                // --- STATE_NEXT folded into this scan (2026-09-02) --------------
                // Saves one PLC scan per recipe line: the line advance no longer
                // costs its own scan. Body is identical to state 60, which STAYS in
                // place -- ten other states still transition to it.
                //
                // MUST stay below the Error / tonMoveTimeout block above, and MUST
                // keep the #state = STATE_NEXT guard: those branches write
                // STATE_ERROR, and the guard is what lets them win. Removing either
                // makes a faulted axis advance the line instead of stopping.
                // See docs/RecipeHandler_ScanLatency.md.
                IF #state = STATE_NEXT THEN
                    #lineIndex := #lineIndex + 1;
                    IF "DB_HMI".SingleStepMode THEN
                        #state := STATE_STEP_WAIT;
                    ELSE
                        #state := STATE_READ;
                    END_IF;
                END_IF;
            END_IF;

        // -----------------------------------------------------------------
        // === STATE_VEL_WAIT (32) -- EXPERIMENTAL velocity-mode segment ===
        // -----------------------------------------------------------------
        // The axes are moving under MC_MoveVelocity toward #targX/#targZ. Nothing
        // here ends in v = 0: when the remaining distance drops under vmSwitchDist
        // the line is counted done and STATE_READ launches the next one (EXEC
        // computes its vector from the ACTUAL position, so the lag of that scan is
        // corrected on the next segment instead of accumulating).
        //
        // Guard order matters: Pause first (operator intent), then run permission,
        // then faults, then completion. Every exit except completion drops
        // vmActive AND brings in a halt, because MC_MoveVelocity keeps running
        // when Execute drops.
        //
        // Fault exits set vmHaltReq THEMSELVES (2026-09-15). "Going to STATE_ERROR"
        // is NOT a halt in the scan it happens: the ERROR branch that sets bHaltTrig
        // only runs on the NEXT scan, so the axes used to keep the stale vector for a
        // whole extra scan after the guard had already fired. The MC_Halt calls sit
        // below the state machine, so vmHaltReq set here reaches the TO in the same
        // scan the velocity command drops. Same rule for the fault branches in the
        // STATE_EXEC launch block. Never remove those lines as "redundant with ERROR".
        32: // VEL_WAIT
            #bTrigMove := FALSE;
            #actX := #Axis_X.ActualPosition;
            #actZ := #Axis_Z.ActualPosition;
            #vmRem := (#targX - #actX) * #vmUX + (#targZ - #actZ) * #vmUZ;
            #vmLat := ABS((#targX - #actX) * #vmUZ - (#targZ - #actZ) * #vmUX);

            IF #Pause THEN
                #vmActive := FALSE;
                #bHaltTrig := TRUE;
                // STATE_PAUSED waits for halt Done only on axes flagged as moving.
                #bMoveX := TRUE;
                #bMoveZ := TRUE;
                // Resume re-reads the line and EXEC relaunches from the interruption
                // point -- same path as a pause taken in STATE_WAIT.
                #pauseReturnState := STATE_READ;
                #state := STATE_PAUSED;

            ELSIF NOT #Start THEN
                // FB_Process left RUNNING without Stop/Pause/Reset reaching us
                // (e.g. its own ERROR). A position move would just finish; a
                // velocity command would not, so stop here.
                #vmActive := FALSE;
                #vmHaltReq := TRUE;   // halt THIS scan -- see the VEL_WAIT header
                #ErrorID := 16#000F;
                "DB_Diagnostic".Error_Text := 'Velocity path: run permission lost';
                "DB_HMI".ErrorDetail := CONCAT(IN1 := 'Ln:', IN2 := CONCAT(
                                        IN1 := INT_TO_STRING(#lineIndex), IN2 := ' run permission lost'));
                #state := STATE_ERROR;

            ELSIF #vmErr THEN
                #vmActive := FALSE;
                #vmHaltReq := TRUE;   // halt THIS scan -- see the VEL_WAIT header
                IF (#vmUseB AND #mcVelXB.Error) OR (NOT #vmUseB AND #mcVelXA.Error) THEN
                    #ErrorID := 16#0001;
                    IF #vmUseB THEN
                        "DB_Diagnostic".MoveX_ErrorID := #mcVelXB.ErrorID;
                    ELSE
                        "DB_Diagnostic".MoveX_ErrorID := #mcVelXA.ErrorID;
                    END_IF;
                    "DB_Diagnostic".TO_ErrorText := "FC_TO_ErrorText"(Code := "DB_Diagnostic".MoveX_ErrorID);
                    "DB_Diagnostic".Error_Text := CONCAT(IN1 := 'X velocity move failed: ', IN2 := "DB_Diagnostic".TO_ErrorText);
                ELSE
                    #ErrorID := 16#0002;
                    IF #vmUseB THEN
                        "DB_Diagnostic".MoveZ_ErrorID := #mcVelZB.ErrorID;
                    ELSE
                        "DB_Diagnostic".MoveZ_ErrorID := #mcVelZA.ErrorID;
                    END_IF;
                    "DB_Diagnostic".TO_ErrorText := "FC_TO_ErrorText"(Code := "DB_Diagnostic".MoveZ_ErrorID);
                    "DB_Diagnostic".Error_Text := CONCAT(IN1 := 'Z velocity move failed: ', IN2 := "DB_Diagnostic".TO_ErrorText);
                END_IF;
                // Single-writer: HMI error from FB_AlarmManager (FB_Process forwards #ErrorID)
                "DB_HMI".ErrorDetail := CONCAT(IN1 := 'Ln:', IN2 := CONCAT(
                                        IN1 := INT_TO_STRING(#lineIndex), IN2 := CONCAT(
                                        IN1 := ' TO:', IN2 := "DB_Diagnostic".TO_ErrorText)));
                #state := STATE_ERROR;

            ELSIF #vmAborted THEN
                // Another motion command took the axis (FB_Process PNP halt, a manual
                // command, ...). Do NOT carry on to the next line -- that would
                // relaunch motion straight through whatever stopped it.
                #vmActive := FALSE;
                #vmHaltReq := TRUE;   // halt THIS scan -- see the VEL_WAIT header
                #ErrorID := 16#000F;
                "DB_Diagnostic".Error_Text := 'Velocity path: aborted by another motion command';
                "DB_HMI".ErrorDetail := CONCAT(IN1 := 'Ln:', IN2 := CONCAT(
                                        IN1 := INT_TO_STRING(#lineIndex), IN2 := ' velocity cmd aborted'));
                #state := STATE_ERROR;

            ELSIF #vmLat > #vmMaxDev
               OR #vmRem > #vmSegLen + #vmMaxDev THEN
                // Off the line, or moving AWAY from the end point. Either means the
                // commanded vector is not what the axes are doing.
                #vmActive := FALSE;
                #vmHaltReq := TRUE;   // halt THIS scan -- see the VEL_WAIT header
                #ErrorID := 16#000F;
                "DB_Diagnostic".Error_Text := CONCAT(IN1 := 'Velocity path deviation mm: ',
                                              IN2 := CONCAT(IN1 := REAL_TO_STRING(MAX(IN1 := #vmLat, IN2 := #vmRem - #vmSegLen)),
                                              IN2 := CONCAT(IN1 := ' limit ', IN2 := REAL_TO_STRING(#vmMaxDev))));
                "DB_HMI".ErrorDetail := CONCAT(IN1 := 'Ln:', IN2 := CONCAT(
                                        IN1 := INT_TO_STRING(#lineIndex), IN2 := ' off path'));
                #state := STATE_ERROR;

            ELSIF #tonMoveTimeout.Q THEN
                #vmActive := FALSE;
                #vmHaltReq := TRUE;   // halt THIS scan -- see the VEL_WAIT header
                #ErrorID := 16#0008;
                "DB_Diagnostic".Error_Text := 'Motion Timeout: velocity path';
                "DB_HMI".ErrorDetail := CONCAT(IN1 := 'Vel path no progress - Ln:',
                                        IN2 := INT_TO_STRING(#lineIndex));
                #state := STATE_ERROR;

            ELSIF #vmRem <= #vmSwitchDist THEN
                // Segment done. The axes keep their current velocity for the scan it
                // takes READ/EXEC to launch the next line -- no halt, no stop.
                // SingleStepMode is deliberately NOT honoured here (the axes are
                // moving). EXEC refuses velocity mode while it is on, so the next line
                // lands with MC_MoveAbsolute and single-step takes over from there.
                #currX := #targX;
                #currZ := #targZ;
                #lineIndex := #lineIndex + 1;
                #state := STATE_READ;
            END_IF;

        // -----------------------------------------------------------------
        // === STATE_TOOL_REQ (40) ===
        // -----------------------------------------------------------------
        40: // TOOL_REQ
            #ToolChangeReq := TRUE;
            #state := STATE_TOOL_WAIT;

        // -----------------------------------------------------------------
        // === STATE_TOOL_WAIT (50) ===
        // -----------------------------------------------------------------
        50: // TOOL_WAIT
            // Wait for external tool change completion from FB_Process
            // FB_Process sets ToolChangeReq := FALSE when done
            // BUG FIX: also wait for Start (bStartSeq) to be TRUE before advancing.
            // Without this, the recipe races ahead through READ→SPINDLE while the machine
            // is still in STATE_LOCK_EXTEND_WAIT (17) where bStartSeq=FALSE.
            // The spindle-start latch is only checked in CASE 20 (RUNNING), so any
            // SpindleReqStart pulse that fires in state 17 is silently missed.
            IF NOT #ToolChangeReq AND #Start THEN
                #state := STATE_NEXT;
            END_IF;

        // -----------------------------------------------------------------
        // === STATE_SPINDLE (55) ===
        // -----------------------------------------------------------------
        55: // SPINDLE -- Forward spindle command to FB_Process (via flag)
            IF #Lines[#lineIndex].CMD = CMD_SPINDLE_ON THEN
                #SpindleReqStart := TRUE;
                #SpindleReqStop := FALSE;
                #SpindleReqSpeed := INT_TO_REAL(BYTE_TO_INT(#Lines[#lineIndex].Param)) * SPINDLE_PARAM_TO_RPM;
                #tonAtSpeed(IN := FALSE, PT := "DB_MachineConfig".Timeout_SpindleAtSpeed);  // reset timer before waiting
                #state := STATE_SPINDLE_WAIT;           // wait for AtSpeed before next motion
            ELSE
                #SpindleReqStart := FALSE;
                #SpindleReqStop := TRUE;
                #SpindleReqSpeed := 0.0;
                #tonAtSpeed(IN := FALSE, PT := "DB_MachineConfig".Timeout_SpindleStop);  // reset timer for stop wait
                #state := STATE_SPINDLE_STOP_WAIT;      // wait for full stop before tool change / next motion
            END_IF;

        // -----------------------------------------------------------------
        // === STATE_SPINDLE_WAIT (56) ===
        // -----------------------------------------------------------------
        56: // SPINDLE_WAIT -- Wait for spindle to reach commanded speed (AtSpeed)
            // DB_Spindle.AtSpeed = TRUE when actual speed is within SpeedTolerance % of commanded.
            // Timeout 10s: error 16#030A. Adjust DB_Spindle.SpeedTolerance if triggering too early.
            // BUG FIX: Clear SpindleReqStart here (one scan after state 55 set it) so it is a
            // true one-shot flag. Without this, FB_Process re-sets bSpindleStart=TRUE every scan
            // because SpindleReqStart was never cleared, preventing FB_SpindleControl from ever
            // seeing a FALSE on its Start input and therefore never generating a rising startEdge.
            #SpindleReqStart := FALSE;
            #tonAtSpeed(IN := TRUE, PT := "DB_MachineConfig".Timeout_SpindleAtSpeed);
            IF "DB_Spindle".AtSpeed OR "DB_Spindle".Bypass_AtSpeed THEN
                #tonAtSpeed(IN := FALSE, PT := "DB_MachineConfig".Timeout_SpindleAtSpeed);  // reset for next use
                #state := STATE_NEXT;
            ELSIF #tonAtSpeed.Q THEN
                #tonAtSpeed(IN := FALSE, PT := "DB_MachineConfig".Timeout_SpindleAtSpeed);  // reset
                #ErrorID := 16#030A;
                "DB_Diagnostic".Error_Text := 'Spindle did not reach target speed (timeout)';
                "DB_Diagnostic".Error_Line := #lineIndex;
                "DB_Diagnostic".Error_Code := #ErrorID;
                // Single-writer: HMI error from FB_AlarmManager (FB_Process forwards #ErrorID)
                "DB_HMI".ErrorDetail    := CONCAT(IN1 := 'Ln:', IN2 := CONCAT(
                                          IN1 := INT_TO_STRING(#lineIndex), IN2 := ' (10s limit)'));
                #state := STATE_ERROR;
            ELSIF #Pause THEN
                #tonAtSpeed(IN := FALSE, PT := "DB_MachineConfig".Timeout_SpindleAtSpeed);
                #bHaltTrig := TRUE;
                #pauseReturnState := STATE_SPINDLE_WAIT;  // resume re-waits AtSpeed, NOT a move
                #state := STATE_PAUSED;
            END_IF;

        // -----------------------------------------------------------------
        // === STATE_DWELL (57) ===
        // -----------------------------------------------------------------
        57: // DWELL -- Wait Param*100ms (equivalent to G4 command)
            // Example: Param=10 → 1000ms (1 second) wait.
            // No axis movement during dwell; spindle continues running.
            IF #Pause THEN
                // Pause pressed -- stop timer and go to PAUSED state
                #tonDwell(IN := FALSE, PT := #dwellTime);
                #bHaltTrig := TRUE;
                #pauseReturnState := STATE_DWELL;  // resume restarts the full dwell, NOT a move
                #state := STATE_PAUSED;
            ELSE
                #tonDwell(IN := TRUE, PT := #dwellTime);
                IF #tonDwell.Q THEN
                    #tonDwell(IN := FALSE, PT := #dwellTime); // Reset timer
                    #state := STATE_NEXT;
                END_IF;
            END_IF;

        // -----------------------------------------------------------------
        // === STATE_SPINDLE_STOP_WAIT (58) ===
        // -----------------------------------------------------------------
        58: // SPINDLE_STOP_WAIT -- Wait for spindle to fully stop before continuing.
            // Prevents a tool change (or next motion line) while spindle is still coasting.
            // DB_Spindle.IsRunning goes FALSE when FB_SpindleControl reaches idle state.
            // Timeout 15s → error 16#030B.
            // BUG FIX: Clear SpindleReqStop here (one scan after state 55 set it) so it is a
            // true one-shot flag. Mirrors the SpindleReqStart fix in state 56.
            #SpindleReqStop := FALSE;
            #tonAtSpeed(IN := TRUE, PT := "DB_MachineConfig".Timeout_SpindleStop);
            IF NOT "DB_Spindle".IsRunning THEN
                #tonAtSpeed(IN := FALSE, PT := "DB_MachineConfig".Timeout_SpindleStop);
                #state := STATE_NEXT;
            ELSIF #tonAtSpeed.Q THEN
                #tonAtSpeed(IN := FALSE, PT := "DB_MachineConfig".Timeout_SpindleStop);
                #ErrorID := 16#030B;
                "DB_Diagnostic".Error_Text := 'Spindle did not stop (timeout)';
                "DB_Diagnostic".Error_Line := #lineIndex;
                "DB_Diagnostic".Error_Code := #ErrorID;
                // Single-writer: HMI error from FB_AlarmManager (FB_Process forwards #ErrorID)
                "DB_HMI".ErrorDetail    := CONCAT(IN1 := 'Ln:', IN2 := CONCAT(
                                          IN1 := INT_TO_STRING(#lineIndex), IN2 := ' (15s limit)'));
                #state := STATE_ERROR;
            ELSIF #Pause THEN
                #tonAtSpeed(IN := FALSE, PT := "DB_MachineConfig".Timeout_SpindleStop);
                #bHaltTrig := TRUE;
                #pauseReturnState := STATE_SPINDLE_STOP_WAIT;  // resume re-waits spindle stop, NOT a move
                #state := STATE_PAUSED;
            END_IF;

        // -----------------------------------------------------------------
        // === STATE_CYL_GOTO (70) ===
        // CMD=40: Trigger BackSupport full extension (PositioningMode=0, no ruler).
        // AtSetpoint fires after Timeout_Extend. Param value is ignored.
        // -----------------------------------------------------------------
        70: // STATE_CYL_GOTO
            "DB_Cylinder_BackSupport".Cmd_Extend := TRUE;
            #state := STATE_CYL_GOTO_WAIT;

        // -----------------------------------------------------------------
        // === STATE_CYL_GOTO_WAIT (71) ===
        // CMD=40: Wait for BackSupport AtSetpoint (Mode=0: after Timeout_Extend elapses).
        // Cmd_Extend re-written every scan to hold the extend command.
        // On done: clear Cmd_Extend. NOTE this does NOT de-energise the cylinder -- the FB
        // stays in State 3 and holds Sol_A ON (09:833-835). That is the operator's spec:
        // Sol_A stays energised until CMD=41 P2 latches Cmd_Retract. (The old comment here
        // claimed "5/3 blocked-center holds position", which was wrong for Mode 0: the hold
        // is live pressure, not the blocked centre.)
        // On error: report and go to STATE_ERROR.
        // -----------------------------------------------------------------
        71: // STATE_CYL_GOTO_WAIT
            "DB_Cylinder_BackSupport".Cmd_Extend := TRUE;
            IF #Pause THEN
                // ITEM-39: Pause during BackSupport extension. Clear Cmd_Extend --
                // the 5/3 blocked-centre valve holds position mechanically.
                // Resume re-enters STATE_CYL_GOTO and re-triggers Cmd_Extend.
                "DB_Cylinder_BackSupport".Cmd_Extend := FALSE;
                #bHaltTrig := TRUE;
                #pauseReturnState := STATE_CYL_GOTO;
                #state := STATE_PAUSED;
            ELSIF "DB_Cylinder_BackSupport".AtSetpoint THEN
                "DB_Cylinder_BackSupport".Cmd_Extend := FALSE;  // FB stays in State 3, Sol_A held ON
                #state := STATE_NEXT;
            ELSIF "DB_Cylinder_BackSupport".Error THEN
                "DB_Cylinder_BackSupport".Cmd_Extend := FALSE;
                #ErrorID := 16#0309;
                "DB_Diagnostic".Error_Text := CONCAT(IN1 := 'CMD40 BackSupport cyl error, Param=',
                                              IN2 := INT_TO_STRING(BYTE_TO_INT(#Lines[#lineIndex].Param)));
                "DB_Diagnostic".Error_Line := #lineIndex;
                "DB_Diagnostic".Error_Code := #ErrorID;
                // Single-writer: HMI error from FB_AlarmManager (FB_Process forwards #ErrorID)
                "DB_HMI".ErrorDetail    := CONCAT(IN1 := 'Ln:', IN2 := CONCAT(
                                          IN1 := INT_TO_STRING(#lineIndex), IN2 := ' target not reached'));
                #state := STATE_ERROR;
            END_IF;

        // -----------------------------------------------------------------
        // === STATE_NEXT (60) ===
        // -----------------------------------------------------------------
        60: // NEXT
            #lineIndex := #lineIndex + 1;
            // SingleStepMode: wait for user to press StepNext before continuing
            IF "DB_HMI".SingleStepMode THEN
                #state := STATE_STEP_WAIT;
            ELSE
                #state := STATE_READ;
            END_IF;

        // -----------------------------------------------------------------
        // === STATE_STEP_WAIT (65) ===
        // -----------------------------------------------------------------
        65: // STEP_WAIT - Wait for StepNext pulse in SingleStep mode
            #Paused := TRUE;  // Show as paused in HMI
            IF #rtStepNext THEN
                // User pressed StepNext, continue to next line
                #Paused := FALSE;
                #state := STATE_READ;
            ELSIF NOT "DB_HMI".SingleStepMode THEN
                // SingleStepMode turned off, continue normally
                #Paused := FALSE;
                #prevStepNext := FALSE;  // Clear stale edge -- prevents false trigger when mode re-enabled
                #state := STATE_READ;
            END_IF;

        // -----------------------------------------------------------------
        // === STATE_DONE (99) ===
        // -----------------------------------------------------------------
        99: // DONE
            #Busy := FALSE;
            #Done := TRUE;
            #ToolChangeReq := FALSE;

        // -----------------------------------------------------------------
        // === STATE_PAUSED (800) ===
        // -----------------------------------------------------------------
        // Pause sequence (return-before-resume): 800 halt/capture -> 801 retract ->
        // 802 hold -> 803 return -> pauseReturnState. This FB does not touch the spindle;
        // FB_Process stops it while paused (State=PAUSED) and spins it back up before it
        // releases Pause (drops bPauseActive) here, so 802 -> 803 return only starts once
        // the spindle is back up to speed. See docs/FB_Process_States.md (STATE_PAUSED).
        // Offset/velocity from DB_MachineConfig.
        // -----------------------------------------------------------------
        800: // PAUSED -- fully stop axes, capture interruption point, then retract
            #Paused := TRUE;
            IF NOT (#fbHaltX.Done OR NOT #bMoveX) OR NOT (#fbHaltZ.Done OR NOT #bMoveZ) THEN
                // Axes not yet stopped -- hold halt command
                #bHaltTrig := TRUE;
            ELSE
                // Axes stopped -- release halt, capture return point, arm retract move.
                #bHaltTrig := FALSE;
                #resumeX := #Axis_X.ActualPosition;   // exact interruption point
                #resumeZ := #Axis_Z.ActualPosition;
                // Retract targets = interruption point + operator offset, clamped to soft limits
                // so a pause near home cannot drive an axis past its limit and fault.
                #targX := LIMIT(MN := "DB_MachineConfig".SoftLimit_MinX,
                                IN := #resumeX + "DB_MachineConfig".PauseRetract_X,
                                MX := "DB_MachineConfig".SoftLimit_MaxX);
                #targZ := LIMIT(MN := "DB_MachineConfig".SoftLimit_MinZ,
                                IN := #resumeZ + "DB_MachineConfig".PauseRetract_Z,
                                MX := "DB_MachineConfig".SoftLimit_MaxZ);
                // Both axes are launched on the same bTrigMove edge (same scan) so they
                // START together. Each runs at PauseRetract_Vel independently and finishes
                // when it reaches its own target (they need not arrive together).
                #velX := "DB_MachineConfig".PauseRetract_Vel;
                #velZ := "DB_MachineConfig".PauseRetract_Vel;
                #bMoveX := ABS(#targX - #resumeX) > 0.01;   // skip axis if no net offset
                #bMoveZ := ABS(#targZ - #resumeZ) > 0.01;
                #bTrigMove := FALSE;   // ensure clean FALSE->TRUE edge for fbMove next scan
                #tonPauseMove(IN := FALSE, PT := "DB_MachineConfig".Timeout_Motion);
                #state := STATE_PAUSE_RETRACT;
            END_IF;

        // -----------------------------------------------------------------
        // === STATE_PAUSE_RETRACT (801) ===
        // -----------------------------------------------------------------
        801: // Move to retracted (tool-clear) position. bHaltTrig stays FALSE (no conflict).
            #Paused := TRUE;
            #bTrigMove := TRUE;   // FALSE->TRUE rising edge triggers fbMoveX/fbMoveZ
            IF (#bMoveX AND #fbMoveX.Error) OR (#bMoveZ AND #fbMoveZ.Error) THEN
                "DB_Diagnostic".Error_Line := #lineIndex;
                IF #bMoveX AND #fbMoveX.Error THEN #ErrorID := 16#0001;
                ELSE #ErrorID := 16#0002; END_IF;
                "DB_Diagnostic".Error_Code := #ErrorID;
                "DB_Diagnostic".Error_Text := 'Pause retract move failed';
                #bTrigMove := FALSE;
                #state := STATE_ERROR;
            ELSIF #tonPauseMove.Q THEN
                #ErrorID := 16#0008;
                "DB_Diagnostic".Error_Line := #lineIndex;
                "DB_Diagnostic".Error_Code := #ErrorID;
                "DB_Diagnostic".Error_Text := 'Pause retract timeout';
                #bTrigMove := FALSE;
                #state := STATE_ERROR;
            ELSIF (NOT #bMoveX OR #fbMoveX.Done) AND (NOT #bMoveZ OR #fbMoveZ.Done) THEN
                #bTrigMove := FALSE;   // drop so a fresh edge can start the return move
                #currX := #targX;      // handler now tracks the retracted position
                #currZ := #targZ;
                #state := STATE_PAUSE_HOLD;
            END_IF;

        // -----------------------------------------------------------------
        // === STATE_PAUSE_HOLD (802) ===
        // -----------------------------------------------------------------
        802: // Held at retracted position. Wait for Continue (Pause released).
            #Paused := TRUE;
            #bTrigMove := FALSE;
            IF NOT #Pause THEN
                // Arm the return move back to the exact interruption point.
                // Both axes launched on the same bTrigMove edge (start together).
                #targX := #resumeX;
                #targZ := #resumeZ;
                #velX := "DB_MachineConfig".PauseRetract_Vel;
                #velZ := "DB_MachineConfig".PauseRetract_Vel;
                #bMoveX := ABS(#targX - #Axis_X.ActualPosition) > 0.01;
                #bMoveZ := ABS(#targZ - #Axis_Z.ActualPosition) > 0.01;
                #bTrigMove := FALSE;   // clean edge next scan
                #tonPauseMove(IN := FALSE, PT := "DB_MachineConfig".Timeout_Motion);
                #state := STATE_PAUSE_RETURN;
            END_IF;

        // -----------------------------------------------------------------
        // === STATE_PAUSE_RETURN (803) ===
        // -----------------------------------------------------------------
        803: // Move back to the interruption point, then resume the original toolpath.
            #Paused := TRUE;
            #bTrigMove := TRUE;
            IF (#bMoveX AND #fbMoveX.Error) OR (#bMoveZ AND #fbMoveZ.Error) THEN
                "DB_Diagnostic".Error_Line := #lineIndex;
                IF #bMoveX AND #fbMoveX.Error THEN #ErrorID := 16#0001;
                ELSE #ErrorID := 16#0002; END_IF;
                "DB_Diagnostic".Error_Code := #ErrorID;
                "DB_Diagnostic".Error_Text := 'Pause return move failed';
                #bTrigMove := FALSE;
                #state := STATE_ERROR;
            ELSIF #tonPauseMove.Q THEN
                #ErrorID := 16#0008;
                "DB_Diagnostic".Error_Line := #lineIndex;
                "DB_Diagnostic".Error_Code := #ErrorID;
                "DB_Diagnostic".Error_Text := 'Pause return timeout';
                #bTrigMove := FALSE;
                #state := STATE_ERROR;
            ELSIF (NOT #bMoveX OR #fbMoveX.Done) AND (NOT #bMoveZ OR #fbMoveZ.Done) THEN
                #bTrigMove := FALSE;
                #Paused := FALSE;
                #currX := #resumeX;    // back on the original path
                #currZ := #resumeZ;
                // Resume the state the pause was taken from. Motion pauses resume via
                // STATE_READ (re-read line endpoint, then EXEC recalculates the remaining
                // move from currX/currZ); dwell/spindle-wait continue in place.
                #state := #pauseReturnState;
            END_IF;

        // -----------------------------------------------------------------
        // === STATE_STOPPING (850) ===
        // -----------------------------------------------------------------
        850: // STOPPING -- Halt active, waiting for both axes to fully stop
            // fbHaltX and fbHaltZ continue to be called with Execute=TRUE.
            // When both return Done, bHaltTrig=FALSE and STATE_DONE is entered.
            // This allows STATE_STOPPING (18) in FB_Process to safely see Busy=FALSE.
            #bHaltTrig := TRUE;
            IF #fbHaltX.Done AND #fbHaltZ.Done THEN
                #bHaltTrig := FALSE;
                #Busy  := FALSE;
                #Done  := TRUE;
                #Paused := FALSE;
                #state := STATE_DONE;
            END_IF;

        // -----------------------------------------------------------------
        // === STATE_ERROR (999) ===
        // -----------------------------------------------------------------
        999: // ERROR
            #Error := TRUE;
            #Busy := FALSE;
            #ToolChangeReq := FALSE;
            #bTrigMove := FALSE;  // Stop move commands -- prevent other axis from running free
            #bMoveX := FALSE;
            #bMoveZ := FALSE;
            #bHaltTrig := TRUE;   // Safely stop both axes (was FALSE -- BUG FIX)
            #vmActive := FALSE;   // Velocity mode: release the command; the halt above stops the axes
            // Ensure diagnostic block contains the latest recipe error context
            // Error_ProcessState is NOT written here (removed 2026-08-17): #state is this
            // FB's own state number, a different numbering space from FB_Process's, and in
            // this branch it is always 999 anyway. It read as a nonsense process state.
            // FB_Process captures the real one at alarm time.
            "DB_Diagnostic".Error_Code := #ErrorID;
            "DB_Diagnostic".Error_Line := #lineIndex;
    END_CASE;

    // -------------------------------------------------------------------------
    // === STATE_EXEC (20) -- deliberately OUTSIDE the CASE above ===
    // -------------------------------------------------------------------------
    // Hoisted 2026-09-02 so a motion line selected by STATE_READ in this scan is
    // also LAUNCHED in this scan, saving one PLC scan per recipe line.
    //
    // MUST stay AFTER the CASE and BEFORE the fbMove calls below. Above the CASE
    // it would run a scan early; below the fbMove calls the Execute edge it sets
    // would not reach MC_MoveAbsolute until the next scan -- both give the scan
    // back, and the second does it silently.
    //
    // Only the CMD_RAPID / CMD_LINEAR / CMD_LINEAR_CONT branch of STATE_READ sets state 20, so every
    // non-motion CMD still gets its own scan. That is required, not incidental:
    // STATE_READ writes the BackSupport solenoid flags directly for CMD_ATMO, and
    // two recipe lines sharing a scan would collide.
    //
    // The other way in is #state := #pauseReturnState (STATE_PAUSE_RETURN, 803).
    // All five pause sites set that variable explicitly and none sets STATE_EXEC;
    // if one ever did, this block would run in the same scan 803 clears bTrigMove,
    // destroying the Execute edge and leaving the axis dead after Continue. The
    // declaration default and the Reset clear were repointed at STATE_READ in this
    // commit for exactly that reason.
    //
    // Full argument: docs/RecipeHandler_ScanLatency.md
    // -------------------------------------------------------------------------
    IF #state = STATE_EXEC THEN
        // --- Velocity mode (EXPERIMENTAL) -- is this line part of a run? ---------
        // The CAM decides: only a CMD_LINEAR_CONT (CMD=2) line with a real feed whose
        // NEXT line is a G1 (CMD=1 or 2) with a real feed. CMD=2 is permission, not a
        // promise -- before a rapid, a marker, a cylinder/spindle/tool line or the end it
        // still lands exactly. CMD=1, rapids, single-step and VelPath_Enable = FALSE all
        // use the MC_MoveAbsolute path below and end exactly on the programmed point, so
        // a recipe without CMD=2 behaves exactly as before whatever the flag says.
        #vmEligible := FALSE;
        IF "DB_MachineConfig".VelPath_Enable AND #Start AND NOT "DB_HMI".SingleStepMode
           AND #Lines[#lineIndex].CMD = CMD_LINEAR_CONT AND #Lines[#lineIndex].F > 0
           AND #lineIndex + 1 < #LineCount THEN
            // Nested, not one expression: SCL evaluates every operand of AND, and
            // #Lines[#lineIndex + 1] on the last line would index past the array.
            IF (#Lines[#lineIndex + 1].CMD = CMD_LINEAR OR #Lines[#lineIndex + 1].CMD = CMD_LINEAR_CONT)
               AND #Lines[#lineIndex + 1].F > 0 THEN
                #vmEligible := TRUE;
            END_IF;
        END_IF;

        // --- Same-scan catch-up (2026-09-14) -------------------------------------
        // With a slow scan and short chords (first real exports: 0.4 mm chords, 0.5 mm of
        // travel per 100 ms scan) the axes can already be past this line's end point, and
        // past the next one too. Skipping ONE passed line per scan was simulated on the
        // real program 2 and was NOT enough: the axes kept an old heading while the curve
        // bent away (0.77 mm off path, and a 16#000F fault in pass 1). Skipping ALL passed
        // lines in the same scan and aiming at the first point genuinely ahead gave 0.023 mm
        // and no reversals (tools/sim_velocity_path.py, docs/MotionSmoothing.md 9.2).
        //
        // "Passed" is measured along the PROGRAMMED segment (currX/currZ = previous
        // programmed end point), so it does not depend on how late the last hand-off was.
        // A line is skipped only INTO a line that is itself velocity-eligible, so the
        // loop can never swallow the hand-over line of a run. Off the programmed line by
        // more than VelPath_MaxDeviation -> EXIT, and the fault branch below fires on the
        // same line. Everything below this block (feed, vector) uses the updated line.
        #vmSkipCount := 0;
        IF #vmEligible AND #vmActive AND NOT (#vmErr OR #vmAborted) THEN
            #vmLeadDist := SQRT(#vmVelX * #vmVelX + #vmVelZ * #vmVelZ) * "DB_MachineConfig".VelPath_LeadTime;
            FOR #vmLoop := 1 TO VM_CATCHUP_MAX DO
                #vmNDX := #targX - #currX;
                #vmNDZ := #targZ - #currZ;
                #vmNLen := SQRT(#vmNDX * #vmNDX + #vmNDZ * #vmNDZ);
                IF #vmNLen <= 0.01 THEN
                    EXIT;   // degenerate line -- handled by the launch branch below
                END_IF;
                #vmDX := #targX - #Axis_X.ActualPosition;
                #vmDZ := #targZ - #Axis_Z.ActualPosition;
                #vmAhead := (#vmDX * #vmNDX + #vmDZ * #vmNDZ) / #vmNLen;
                #vmNLat := ABS(#vmDX * #vmNDZ - #vmDZ * #vmNDX) / #vmNLen;
                IF #vmNLat > #vmMaxDev OR #vmAhead > #vmLeadDist THEN
                    EXIT;
                END_IF;
                // Is the NEXT line velocity-eligible? Nested so no index past LineCount is read.
                #vmNextOK := FALSE;
                IF #lineIndex + 2 < #LineCount THEN
                    IF #Lines[#lineIndex + 1].CMD = CMD_LINEAR_CONT AND #Lines[#lineIndex + 1].F > 0 THEN
                        IF (#Lines[#lineIndex + 2].CMD = CMD_LINEAR OR #Lines[#lineIndex + 2].CMD = CMD_LINEAR_CONT)
                           AND #Lines[#lineIndex + 2].F > 0 THEN
                            #vmNextOK := TRUE;
                        END_IF;
                    END_IF;
                END_IF;
                IF NOT #vmNextOK THEN
                    EXIT;   // last line before the hand-over: the single skip below handles it
                END_IF;
                #currX := #targX;
                #currZ := #targZ;
                #lineIndex := #lineIndex + 1;
                #vmSkipCount := #vmSkipCount + 1;
                #targX := #Lines[#lineIndex].X;
                #targZ := #Lines[#lineIndex].Z;
            END_FOR;
        END_IF;

        // Leaving a velocity run: plan the MC_MoveAbsolute from where the axes really
        // are (currX/currZ hold the previous NOMINAL end point), and command BOTH
        // axes below -- an axis with < 0.01 mm left but a live velocity would
        // otherwise never be told to stop.
        #vmWasActive := #vmActive AND NOT #vmEligible;
        IF #vmWasActive THEN
            #currX := #Axis_X.ActualPosition;
            #currZ := #Axis_Z.ActualPosition;
            #vmActive := FALSE;
        END_IF;

        // Linear interpolation: both axes start and finish simultaneously.
        // velX/velZ split proportionally over total distance.
        // This ensures X and Z reach target in the same time (true linear path).
        #deltaX := ABS(#targX - #currX);
        #deltaZ := ABS(#targZ - #currZ);
        #totalDist := SQRT(#deltaX * #deltaX + #deltaZ * #deltaZ);

        // Determine which axes need to move
        #bMoveX := #deltaX > 0.01;  // 0.01mm threshold
        #bMoveZ := #deltaZ > 0.01;
        IF #vmWasActive THEN
            #bMoveX := TRUE;   // see the hand-over comment above
            #bMoveZ := TRUE;
        END_IF;

        // Calculate velocity
        IF #Lines[#lineIndex].CMD = CMD_RAPID OR #Lines[#lineIndex].F = 0 THEN
            // Rapid move - use max velocity with RapidOverride
            #feedrate := "DB_MachineConfig".RapidVelocity;
            #overridePercent := "DB_HMI".RapidOverride;
        ELSE
            // Linear move - convert mm/min to mm/s with FeedrateOverride
            #feedrate := INT_TO_REAL(#Lines[#lineIndex].F) / "DB_MachineConfig".FeedrateConvFactor;
            #overridePercent := "DB_HMI".FeedrateOverride;
        END_IF;

        // Apply override (clamp to 50-200%)
        IF #overridePercent < 50.0 THEN #overridePercent := 50.0; END_IF;
        IF #overridePercent > 200.0 THEN #overridePercent := 200.0; END_IF;
        #feedrate := #feedrate * (#overridePercent / 100.0);

        // Clamp velocity to limits
        IF #feedrate > "DB_MachineConfig".MaxVelocity THEN
            #feedrate := "DB_MachineConfig".MaxVelocity;
        ELSIF #feedrate < "DB_MachineConfig".MinVelocity THEN
            #feedrate := "DB_MachineConfig".MinVelocity;
        END_IF;

        // Calculate axis velocities for linear interpolation
        IF #totalDist > 0.01 THEN
            #velX := #feedrate * #deltaX / #totalDist;
            #velZ := #feedrate * #deltaZ / #totalDist;
        ELSE
            #velX := #feedrate;
            #velZ := #feedrate;
        END_IF;

        // Hand-over speed floor (2026-09-25, narrowed 2026-09-29). The proportional split
        // above assumes both axes start from standstill. At a hand-over they are still
        // moving, and an axis with almost nothing left (program 1 line 197, 2026-09-24
        // export: X-only CMD=1 link, Z ~0..0.2 mm left at 4.4 mm/s) got a crawl speed,
        // down to MinVelocity. It could not stop in the distance left, overshot, and crept
        // back at that crawl speed -- the 2-3 s wait at pass ends. The floor (never slower
        // than the live speed, capped at this line's feed) fixed that.
        //
        // But applied to EVERY hand-over it broke long ending lines: program 1 line 35
        // (2026-09-29 export, 93 mm) had Z forced from 3.5 to 7 mm/s, Z arrived 5.6 s
        // early and X then ran the last ~42 mm ALONE -- up to ~17 mm off the path, the
        // "X move at the end of the pass" the operator reported.
        //
        // So the floor applies to an axis ONLY when it is needed:
        //   * its distance left is within its braking distance from the live speed
        //     (it cannot slow to its proportional share in time -> overshoot), or
        //   * its target is BEHIND it (it must reverse; the return must not crawl).
        // Otherwise the axis gets its proportional share and slows to it in well under
        // a millimetre, finishing together with the other axis. A floored axis can only
        // finish early by at most its braking distance (~0.8 mm at 4.4 mm/s, ~4 mm at
        // F1000), not by the whole line.
        //
        // Never remove the floor as "breaks linear interpolation" (the crawl comes back),
        // and never widen it back to every hand-over (the long-line error comes back).
        // Offline check of both: tools/split_recipe_db.py (hand-over report).
        IF #vmWasActive THEN
            #vmBrakeV := ABS(#vmVelX);
            IF #vmBrakeV <= VM_HO_DEC * VM_HO_DEC / VM_HO_JERK THEN
                #vmBrakeX := #vmBrakeV * SQRT(#vmBrakeV / VM_HO_JERK);   // S-curve, decel never saturates
            ELSE
                #vmBrakeX := #vmBrakeV * #vmBrakeV / (2.0 * VM_HO_DEC) + #vmBrakeV * VM_HO_DEC / (2.0 * VM_HO_JERK);
            END_IF;
            #vmBrakeX := VM_HO_MARGIN * (#vmBrakeX + #vmBrakeV * VM_HO_SCAN);

            #vmBrakeV := ABS(#vmVelZ);
            IF #vmBrakeV <= VM_HO_DEC * VM_HO_DEC / VM_HO_JERK THEN
                #vmBrakeZ := #vmBrakeV * SQRT(#vmBrakeV / VM_HO_JERK);
            ELSE
                #vmBrakeZ := #vmBrakeV * #vmBrakeV / (2.0 * VM_HO_DEC) + #vmBrakeV * VM_HO_DEC / (2.0 * VM_HO_JERK);
            END_IF;
            #vmBrakeZ := VM_HO_MARGIN * (#vmBrakeZ + #vmBrakeV * VM_HO_SCAN);

            // currX/currZ hold the ACTUAL position here (set in the hand-over block above).
            IF #deltaX <= #vmBrakeX OR (#targX - #currX) * #vmVelX < 0.0 THEN
                #velX := MAX(IN1 := #velX, IN2 := MIN(IN1 := ABS(#vmVelX), IN2 := #feedrate));
            END_IF;
            IF #deltaZ <= #vmBrakeZ OR (#targZ - #currZ) * #vmVelZ < 0.0 THEN
                #velZ := MAX(IN1 := #velZ, IN2 := MIN(IN1 := ABS(#vmVelZ), IN2 := #feedrate));
            END_IF;
        END_IF;

        // Ensure minimum velocity
        IF #bMoveX AND #velX < "DB_MachineConfig".MinVelocity THEN
            #velX := "DB_MachineConfig".MinVelocity;
        END_IF;
        IF #bMoveZ AND #velZ < "DB_MachineConfig".MinVelocity THEN
            #velZ := "DB_MachineConfig".MinVelocity;
        END_IF;

        IF #vmEligible THEN
            // --- Velocity-mode launch -------------------------------------------
            // Vector from the ACTUAL position, not from currX/currZ: whatever the
            // previous segment over- or under-ran is absorbed here.
            #actX := #Axis_X.ActualPosition;
            #actZ := #Axis_Z.ActualPosition;
            #vmDX := #targX - #actX;
            #vmDZ := #targZ - #actZ;
            #vmDist := SQRT(#vmDX * #vmDX + #vmDZ * #vmDZ);
            // Lead distance, capped at HALF the segment. The cap is what keeps a slow
            // scan safe: at a ~100 ms OB1 cycle and 5 mm/s the uncapped lead can exceed
            // a whole 1 mm chord, and every line would then be "done" on arrival.
            #vmSwitchDist := MIN(IN1 := #feedrate * "DB_MachineConfig".VelPath_LeadTime,
                                 IN2 := 0.5 * #vmDist);

            // Short-segment catch-up (2026-09-14). With a slow scan a short line (the
            // first real exports have 0.4 mm chords at 5 mm/s = 0.5 mm per 100 ms scan) can
            // be over before the axes are even commanded toward it. Aiming from the actual
            // position at an end point that is already BEHIND the axes would pull them
            // backwards and zig-zag. So measure progress along the PROGRAMMED segment
            // (currX/currZ = previous programmed end point), independent of how late the
            // last hand-off was, and treat a passed end point as done.
            #vmNDX := #targX - #currX;
            #vmNDZ := #targZ - #currZ;
            #vmNLen := SQRT(#vmNDX * #vmNDX + #vmNDZ * #vmNDZ);
            IF #vmNLen > 0.01 THEN
                #vmAhead := (#vmDX * #vmNDX + #vmDZ * #vmNDZ) / #vmNLen;
                #vmNLat := ABS(#vmDX * #vmNDZ - #vmDZ * #vmNDX) / #vmNLen;
            ELSE
                #vmAhead := 0.0;
                #vmNLat := 0.0;
            END_IF;
            #vmSkipDist := MIN(IN1 := #feedrate * "DB_MachineConfig".VelPath_LeadTime,
                               IN2 := 0.5 * #vmNLen);

            IF #vmActive AND (#vmErr OR #vmAborted) THEN
                // The live command died between VEL_WAIT's last check and this scan.
                #vmActive := FALSE;
                #vmHaltReq := TRUE;   // halt THIS scan -- see the VEL_WAIT header
                #ErrorID := 16#000F;
                "DB_Diagnostic".Error_Text := 'Velocity path: command lost between segments';
                "DB_HMI".ErrorDetail := CONCAT(IN1 := 'Ln:', IN2 := CONCAT(
                                        IN1 := INT_TO_STRING(#lineIndex), IN2 := ' velocity cmd lost'));
                #state := STATE_ERROR;
            ELSIF #vmDist <= 0.01 OR #vmNLen <= 0.01 THEN
                // Degenerate line (end point already reached). Take the next line on the
                // NEXT scan via STATE_READ -- not STATE_NEXT, which costs a second scan.
                //
                // This used to skip every line shorter than the lead distance. With a slow
                // scan that skip could chain: each skipped line costs scans, the axes run on
                // the stale vector meanwhile, and VEL_WAIT's deviation guard never runs
                // because the state never gets there. A real segment is now always
                // commanded; only a genuinely zero-length line is skipped.
                #currX := #targX;
                #currZ := #targZ;
                #lineIndex := #lineIndex + 1;
                #state := STATE_READ;
            ELSIF #vmActive AND #vmNLat > #vmMaxDev THEN
                // Checked BEFORE the catch-up skip: skipping is only allowed while the axes
                // are still on the programmed path. This is the deviation guard for lines
                // that never reach STATE_VEL_WAIT.
                #vmActive := FALSE;
                #vmHaltReq := TRUE;   // halt THIS scan -- see the VEL_WAIT header
                #ErrorID := 16#000F;
                "DB_Diagnostic".Error_Text := CONCAT(IN1 := 'Velocity path off programmed line mm: ',
                                              IN2 := CONCAT(IN1 := REAL_TO_STRING(#vmNLat),
                                              IN2 := CONCAT(IN1 := ' limit ', IN2 := REAL_TO_STRING(#vmMaxDev))));
                "DB_HMI".ErrorDetail := CONCAT(IN1 := 'Ln:', IN2 := CONCAT(
                                        IN1 := INT_TO_STRING(#lineIndex), IN2 := ' off path (catch-up)'));
                #state := STATE_ERROR;
            ELSIF #vmActive AND #vmSkipCount >= VM_CATCHUP_MAX THEN
                // The catch-up loop used its whole budget in one scan: more than
                // VM_CATCHUP_MAX programmed points lie inside the lead distance. That is a
                // recipe (segment length) problem, not something to ride through one line
                // per scan. Stop. (Real program 2 needed at most 2 at a 100 ms scan.)
                #vmActive := FALSE;
                #vmHaltReq := TRUE;   // halt THIS scan -- see the VEL_WAIT header
                #ErrorID := 16#000F;
                "DB_Diagnostic".Error_Text := 'Velocity path: too many points inside lead distance - check CAM segment length';
                "DB_HMI".ErrorDetail := CONCAT(IN1 := 'Ln:', IN2 := CONCAT(
                                        IN1 := INT_TO_STRING(#lineIndex), IN2 := ' catch-up limit'));
                #state := STATE_ERROR;
            ELSIF #vmActive AND #vmAhead <= #vmSkipDist THEN
                // Axes are already at (or past) this line's end point: count it done and
                // take the next line on the next scan, keeping the current velocity. Never
                // aim backwards. Bounded by geometry -- it can only fire for end points the
                // axes have genuinely reached -- and guarded by the vmNLat test above.
                #currX := #targX;
                #currZ := #targZ;
                #lineIndex := #lineIndex + 1;
                #state := STATE_READ;
            ELSIF #vmActive AND (#vmDX * #vmVelX + #vmDZ * #vmVelZ) < 0.0 THEN
                // NO REVERSAL WITHIN A RUN. The new vector would turn the path more than
                // 90 degrees against the current direction of travel (vmVelX/Z still hold the
                // live command here). Inside a run that never happens on a valid recipe:
                // SpinningCam emits CMD=1 (exact stop) at turns >= its stop angle, default
                // 90 degrees, and a passed point is skipped above. So a velocity command is
                // never allowed to drive the axes back along the path -- stop instead.
                // If the CAM stop angle is ever raised above 90 degrees, this fires on those
                // corners: safe, and the fix is the CAM setting, never removing this branch.
                #vmActive := FALSE;
                #vmHaltReq := TRUE;   // halt THIS scan -- see the VEL_WAIT header
                #ErrorID := 16#000F;
                "DB_Diagnostic".Error_Text := 'Velocity path: next segment would reverse the direction of travel';
                "DB_HMI".ErrorDetail := CONCAT(IN1 := 'Ln:', IN2 := CONCAT(
                                        IN1 := INT_TO_STRING(#lineIndex), IN2 := ' reverse blocked'));
                #state := STATE_ERROR;
            ELSE
                #vmVelX := #feedrate * #vmDX / #vmDist;
                #vmVelZ := #feedrate * #vmDZ / #vmDist;
                // Below the TO start/stop velocity a non-zero command is rejected;
                // an exact 0.0 is the permitted "hold" value.
                IF ABS(#vmVelX) < "DB_MachineConfig".MinVelocity THEN #vmVelX := 0.0; END_IF;
                IF ABS(#vmVelZ) < "DB_MachineConfig".MinVelocity THEN #vmVelZ := 0.0; END_IF;
                #vmUX := #vmDX / #vmDist;
                #vmUZ := #vmDZ / #vmDist;
                #vmSegLen := #vmDist;
                IF #vmActive THEN
                    #vmUseB := NOT #vmUseB;   // same-scan hand-off to the other instance pair
                END_IF;
                #vmActive := TRUE;
                #velX := ABS(#vmVelX);        // diagnostics only
                #velZ := ABS(#vmVelZ);
                #bMoveX := FALSE;             // no MC_MoveAbsolute in this mode
                #bMoveZ := FALSE;
                #tonMoveTimeout(IN := FALSE, PT := "DB_MachineConfig".Timeout_Motion);
                #state := STATE_VEL_WAIT;
            END_IF;
        // Skip if no movement needed
        ELSIF NOT #bMoveX AND NOT #bMoveZ THEN
            #state := STATE_NEXT;
        ELSE
            // Trigger movement
            #bTrigMove := TRUE;
            #tonMoveTimeout(IN := FALSE, PT := "DB_MachineConfig".Timeout_Motion);
            #state := STATE_WAIT;
        END_IF;
    END_IF;

    // -------------------------------------------------------------------------
    // Motion FB calls -- run at end of every scan (after state machine)
    // bTrigMove AND bMoveX/Z: active only in EXEC state and when axis is needed
    // bHaltTrig: TRUE in STOPPING and PAUSED states -- decelerates axis to stop
    // -------------------------------------------------------------------------
    // =========================================================================
    // VELOCITY-MODE SAFETY NET (EXPERIMENTAL) -- every scan, whatever the state
    // =========================================================================
    // MC_MoveVelocity keeps the axes moving until something stops them. Every exit
    // path in the state machine stops them explicitly -- but that is many separate
    // places, and one missed or broken path means an axis driving to its hardware
    // limit. These two checks do not depend on any of those paths being right:
    //
    //   NET 1 (here, BEFORE the motion calls): a velocity command may only be live in
    //         READ / EXEC / VEL_WAIT. In any other state -- however it got there --
    //         drop it and halt. Before the calls, so the dropped Execute and the
    //         halt reach the TO in the same scan.
    //   NET 2 (after the motion calls): a velocity instance still Busy while no
    //         velocity command is supposed to be live, for more than
    //         VM_UNSUPERVISED_SCANS scans -> halt and fault 16#000F. Catches a hand-over
    //         MC_MoveAbsolute that never took over (the handler would otherwise sit in
    //         STATE_WAIT with no path guard for Timeout_Motion), and anything else.
    //
    // DO NOT remove, weaken or move either net behind a state test.
    IF #vmActive AND NOT (#state = STATE_READ OR #state = STATE_EXEC OR #state = STATE_VEL_WAIT) THEN
        #vmActive := FALSE;
        #vmHaltReq := TRUE;
    END_IF;

    #fbMoveX(Execute := #bTrigMove AND #bMoveX, Position := #targX, Velocity := #velX, Axis := #Axis_X);
    #fbMoveZ(Execute := #bTrigMove AND #bMoveZ, Position := #targZ, Velocity := #velZ, Axis := #Axis_Z);
    #fbHaltX(Execute := #bHaltTrig OR #vmHaltReq, Axis := #Axis_X);
    #fbHaltZ(Execute := #bHaltTrig OR #vmHaltReq, Axis := #Axis_Z);

    // Velocity mode (EXPERIMENTAL). Direction := 0 = direction from the sign of
    // Velocity. Exactly one pair has Execute TRUE while vmActive; see the VAR block.
    #mcVelXA(Axis := #Axis_X, Execute := #vmActive AND NOT #vmUseB, Velocity := #vmVelX, Direction := 0);
    #mcVelXB(Axis := #Axis_X, Execute := #vmActive AND #vmUseB, Velocity := #vmVelX, Direction := 0);
    #mcVelZA(Axis := #Axis_Z, Execute := #vmActive AND NOT #vmUseB, Velocity := #vmVelZ, Direction := 0);
    #mcVelZB(Axis := #Axis_Z, Execute := #vmActive AND #vmUseB, Velocity := #vmVelZ, Direction := 0);
    // Status of the LIVE pair, read by VEL_WAIT / EXEC next scan. The pair just
    // switched away from reports CommandAborted by design and is not looked at.
    IF #vmUseB THEN
        #vmErr     := #mcVelXB.Error OR #mcVelZB.Error;
        #vmAborted := #mcVelXB.CommandAborted OR #mcVelZB.CommandAborted;
    ELSE
        #vmErr     := #mcVelXA.Error OR #mcVelZA.Error;
        #vmAborted := #mcVelXA.CommandAborted OR #mcVelZA.CommandAborted;
    END_IF;
    // NET 2 -- unsupervised velocity command (see the safety-net header above the calls).
    IF NOT #vmActive AND (#mcVelXA.Busy OR #mcVelXB.Busy OR #mcVelZA.Busy OR #mcVelZB.Busy) THEN
        #vmUnsupScans := #vmUnsupScans + 1;
    ELSE
        #vmUnsupScans := 0;
    END_IF;
    IF #vmUnsupScans > VM_UNSUPERVISED_SCANS THEN
        #vmHaltReq := TRUE;
        #vmUnsupScans := 0;
        IF #state <> STATE_IDLE AND #state <> STATE_DONE AND #state <> STATE_ERROR THEN
            #ErrorID := 16#000F;
            "DB_Diagnostic".Error_Text := 'Velocity path: velocity command active without supervision - halted';
            "DB_HMI".ErrorDetail := CONCAT(IN1 := 'Ln:', IN2 := CONCAT(
                                    IN1 := INT_TO_STRING(#lineIndex), IN2 := ' unsupervised vel cmd'));
            #state := STATE_ERROR;
        END_IF;
    END_IF;
    // Reset/safety-net halt releases once both axes report the halt Done, OR both are
    // at standstill with no velocity command busy -- the second so a halt that cannot
    // complete (drive already off) can never lock the handler out of the next start.
    IF #vmHaltReq
       AND NOT (#mcVelXA.Busy OR #mcVelXB.Busy OR #mcVelZA.Busy OR #mcVelZB.Busy)
       AND ((#fbHaltX.Done AND #fbHaltZ.Done)
            OR (#Axis_X.StatusBits.StandStill AND #Axis_Z.StatusBits.StandStill)) THEN
        #vmHaltReq := FALSE;
    END_IF;

    // Calculate progress
    IF #LineCount > 0 THEN
        #Progress := INT_TO_REAL(#lineIndex) / INT_TO_REAL(#LineCount) * 100.0;
    ELSE
        #Progress := 0.0;
    END_IF;

    // Update active feedrate for HMI (convert mm/s back to mm/min using same factor as forward conversion)
    #ActiveFeedrate := #feedrate * "DB_MachineConfig".FeedrateConvFactor;

    // Outputs
    #CurrentLine := #lineIndex;

    // Diagnostics
    "DB_Diagnostic".Recipe_CurrentLine := #lineIndex;
    "DB_Diagnostic".Recipe_TargetX := #targX;
    "DB_Diagnostic".Recipe_TargetZ := #targZ;
    "DB_Diagnostic".Recipe_Velocity := #velX;
    "DB_Diagnostic".bMoveX := #bMoveX;
    "DB_Diagnostic".bMoveZ := #bMoveZ;
    "DB_Diagnostic".MoveX_Busy := #fbMoveX.Busy;
    "DB_Diagnostic".MoveX_Done := #fbMoveX.Done;
    "DB_Diagnostic".MoveX_Error := #fbMoveX.Error;
    "DB_Diagnostic".MoveZ_Busy := #fbMoveZ.Busy;
    "DB_Diagnostic".MoveZ_Done := #fbMoveZ.Done;
    "DB_Diagnostic".MoveZ_Error := #fbMoveZ.Error;
END_FUNCTION_BLOCK
